// TwinCAT 3 PLC project TC3_ST_PC2_DistributedTest
// ProgramVersion: 3.1.4023.0
// libraries:
//   DistributedControl, * (FactoryAutomation)
//   Tc2_Standard, * (Beckhoff Automation GmbH)
//   Tc2_System, * (Beckhoff Automation GmbH)
//   Tc3_Module, * (Beckhoff Automation GmbH)
// project tree:
//   / PlcTask.TcTTO
//   POUs/ MAIN.TcPOU
// real-time tasks:
//   TASK PlcTask: cycle T#10ms, priority 22, ADS port 350

CONFIGURATION TC3_ST_PC2_DistributedTest
    RESOURCE PLC ON TwinCAT3
        TASK PlcTask(INTERVAL := T#10ms, PRIORITY := 22);
        PROGRAM MAIN WITH PlcTask : MAIN;
    END_RESOURCE
END_CONFIGURATION

// ---- POUs/MAIN.TcPOU
PROGRAM MAIN
VAR
		
	bStart : BOOL;
	fbPayloadClient : Payload(uiObjectSize := SIZEOF(Payload));
	aClientMarshalBuffer : ARRAY[0..1999] OF BYTE;
	aClientUnmarshalBuffer : ARRAY[0..1999] OF BYTE;
	fbClient : TcpIp(TCP_IP_CLIENT);
	clientStep : UINT;
	udiClientTimeToSend : UDINT;
	udiClientTimeToReceive : UDINT;
	udiClientTimeToSendTmp : UDINT;
	udiClientTimeToReceiveTmp : UDINT;
END_VAR


fbPayloadClient();

fbClient.stClientData.nRemotePort := 200;
fbClient.stClientData.sRemoteHost := '192.168.2.115';
fbClient(bEnable := TRUE);

IF 	bStart
	THEN
	
	
	CASE clientStep OF
	
		0 :
 			IF 	fbClient.ReceiveSerializedObject(pDest := ADR(aClientUnmarshalBuffer),cbLen := fbPayloadClient.uiObjectSize)
				THEN
				
				fbPayloadClient.Deserialize(ADR(aClientUnmarshalBuffer));
				MEMCPY(ADR(aClientMarshalBuffer),fbPayloadClient.Serialize(),fbPayloadClient.uiObjectSize);
				
				clientStep := 10;
				
			END_IF
			
		10: 
			IF 	fbClient.SendSerializedObject(pSrc := ADR(aClientMarshalBuffer), cbLen := fbPayloadClient.uiObjectSize)
				THEN
				
				clientStep := 0;
			END_IF
		
	END_CASE


END_IF

END_PROGRAM
